(* Logix 5000 project; controller DeviceNetTest vendor 1 type 14 code 79 rev 17.4; software revision 17.01 *)

TASK MainTask (continuous, watchdog 500 ms) : MainProgram, DeviceN

MODULES
   Local : vendor 1 type 14 code 79 (ICP 0, rev 17.4)
      DN : vendor 1 type 12 code 14 (ICP 2, rev 7.3, Output RPI 20 ms, Input RPI 20 ms)
      Ethernet : 1756-ENBT (Ethernet 192.168.0.4, ICP 3, rev 4.1)
         Camera_Sensor : ETHERNET-MODULE (Ethernet 192.168.0.3, rev 1.1, Output RPI 100 ms)   // Banner
      LocalSERCOS : vendor 1 type 16 code 14 (ICP 1, rev 17.2, MotionAsync RPI 25 ms, MotionEvent RPI 1000 ms, MotionSync RPI 2 ms)
         Drive : vendor 1 type 115 code 164 (SERCOS 1, rev 1.1)
END_MODULES

VAR_GLOBAL   (* controller tags *)
   botao : BOOL;
   dir_int : DINT;
   direction : BOOL;
   drive_axis : AXIS_SERVO_DRIVE;
   Emanuel : BOOL;
   encoder : AXIS_SERVO_DRIVE;
   MAH_0 : MOTION_INSTRUCTION;
   MAJ_0 : MOTION_INSTRUCTION := (FLAGS := 33554432);
   MAJ_1 : MOTION_INSTRUCTION := (FLAGS := 33554432);
   MAJ_2 : MOTION_INSTRUCTION;
   MAS_0 : MOTION_INSTRUCTION;
   MAS_1 : MOTION_INSTRUCTION := (FLAGS := 33554432);
   MAS_2 : MOTION_INSTRUCTION;
   MGroup : MOTION_GROUP;
   MSF_0 : MOTION_INSTRUCTION;
   MSO_0 : MOTION_INSTRUCTION;
   MSO_1 : MOTION_INSTRUCTION := (FLAGS := -1610612736, EN := 1, DN := 1, STATE := 1);
   timer_1 : TIMER := (PRE := 500);
   trigger_off : TIMER := (PRE := 200);
   trigger_on : TIMER := (PRE := 200);
END_VAR

PROGRAM Camera_Trigger   (* main routine TriggerMain *)
// Trigger
VAR
   Trigger : ALIAS FOR Camera_Sensor:O.Data[0].0;
END_VAR

ROUTINE TriggerMain   (* ladder *)
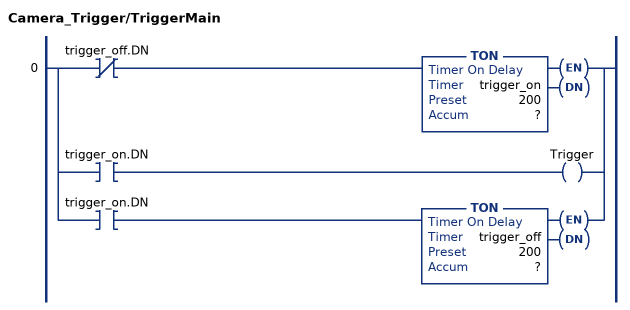
   0: [XIO(trigger_off.DN) TON(trigger_on,?,?) ,XIC(trigger_on.DN) OTE(Trigger) ,XIC(trigger_on.DN) TON(trigger_off,?,?) ];
END_ROUTINE
END_PROGRAM

PROGRAM DeviceN   (* main routine InitDNetST *)

ROUTINE InitDNetST   (* structured text *)
   Local:2:O.CommandRegister.Run [:=] 1;
   
END_ROUTINE
END_PROGRAM

PROGRAM MainProgram   (* main routine MainRoutineST *)

ROUTINE MainRoutine   (* ladder *)
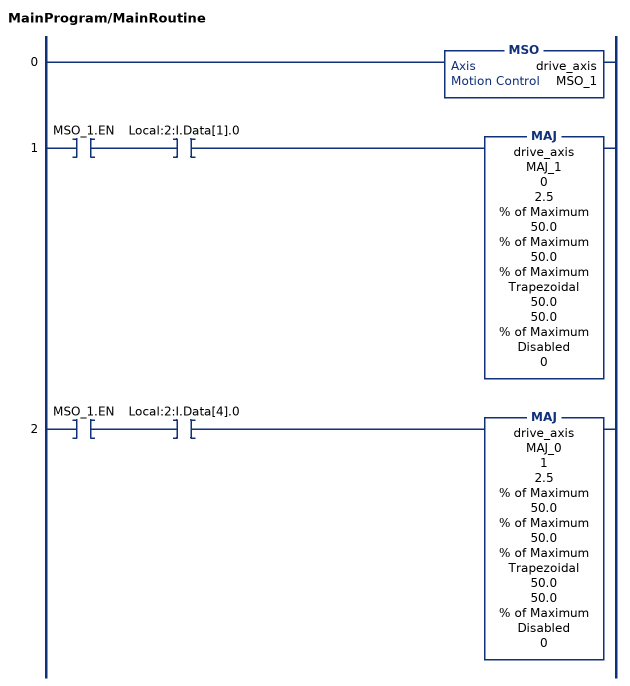
   0: MSO(drive_axis,MSO_1);
   1: XIC(MSO_1.EN)XIC(Local:2:I.Data[1].0)MAJ(drive_axis,MAJ_1,0,2.5,% of Maximum,50.0,% of Maximum,50.0,% of Maximum,Trapezoidal,50.0,50.0,% of Maximum,Disabled,0);
   2: XIC(MSO_1.EN)XIC(Local:2:I.Data[4].0)MAJ(drive_axis,MAJ_0,1,2.5,% of Maximum,50.0,% of Maximum,50.0,% of Maximum,Trapezoidal,50.0,50.0,% of Maximum,Disabled,0);
END_ROUTINE

ROUTINE MainRoutineST   (* structured text *)
   MSO(drive_axis,MSO_1);
   IF MSO_1.EN AND Local:2:I.Data[1].0 THEN
   	MAJ(drive_axis,MAJ_1,0,2.5,1,50.0,1,50.0,1,0,50.0,50.0,1,0,0);
   END_IF;
   IF MSO_1.EN AND Local:2:I.Data[4].0 THEN
   	MAJ(drive_axis,MAJ_0,1,2.5,1,50.0,1,50.0,1,0,50.0,50.0,1,0,0);
   END_IF;
END_ROUTINE
END_PROGRAM

PROGRAM Parada   (* main routine parada *)

ROUTINE parada   (* ladder *)
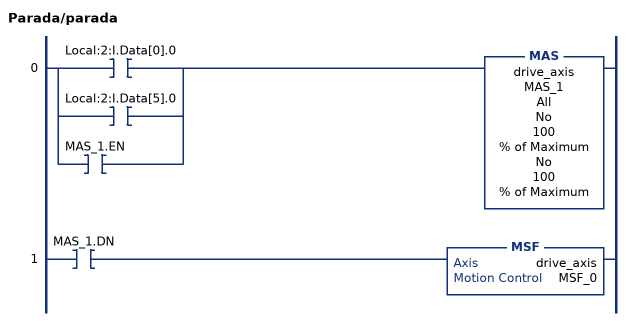
   0: [XIC(Local:2:I.Data[0].0) ,[XIC(Local:2:I.Data[5].0) ,XIC(MAS_1.EN) ] ]MAS(drive_axis,MAS_1,All,No,100,% of Maximum,No,100,% of Maximum);
   1: XIC(MAS_1.DN)MSF(drive_axis,MSF_0);
END_ROUTINE
END_PROGRAM
